FUNCTION_BLOCK FB_HMI_BUTTON
VAR_INPUT
    stColor : T_HMI_COLORS;
END_VAR
VAR_IN_OUT
    nActiveTab : INT;
    sActiveName : STRING;
END_VAR
VAR_OUTPUT
    sName : STRING;
    sIconName : STRING;
    nThisTab : INT;
    bActivated : BOOL;
    bNotActivated : BOOL;
    
    bIsNotGreen : BOOL;
    bIsNotRed : BOOL;
    bIsNotBlue : BOOL;
    bIsNotOrange : BOOL;
    bIsNotGray : BOOL;
END_VAR
VAR
    bDoActivate : BOOL;
    bPreviouslyActive : BOOL;
END_VAR

IF bDoActivate THEN
    nActiveTab := nThisTab;
    bDoActivate := FALSE;
END_IF

bActivated := nActiveTab = nThisTab;
bNotActivated := NOT bActivated;

IF bActivated AND NOT bPreviouslyActive THEN
    sActiveName := sName;
    bPreviouslyActive := TRUE;
END_IF

IF bNotActivated THEN
    bPreviouslyActive := FALSE;
END_IF

bIsNotRed    := stColor.bg <> E_HMI_Colors.RED;
bIsNotBlue   := stColor.bg <> E_HMI_Colors.BLUE;
bIsNotOrange := stColor.bg <> E_HMI_Colors.ORANGE;
bIsNotGray   := stColor.bg <> E_HMI_Colors.GRAY;
bIsNotGreen  := stColor.bg <> E_HMI_Colors.GREEN;

METHOD FB_init : BOOL
VAR_INPUT
	bInitRetains : BOOL; // if TRUE, the retain variables are initialized (warm start / cold start)
	bInCopyCode : BOOL;  // if TRUE, the instance afterwards gets moved into the copy code (online change)
    sName : STRING;
    sIconName : STRING;
    nThisTab : INT;
END_VAR
THIS^.sName := sName;
THIS^.sIconName := sIconName;
THIS^.nThisTab := nThisTab;
END_METHOD

METHOD M_SetIconName
VAR_INPUT
    sIconName : STRING;
END_VAR
THIS^.sIconName := sIconName;
END_METHOD

END_FUNCTION_BLOCK

(* stored: Version 1.1.0.1, ProductVersion 3.1.4024.14
   POU FB_HMI_BUTTON: Id {8312f969-1e2d-4234-8fb1-a5ec8ac8ee74}, SpecialFunc None
   Method FB_init: Id {09c2525c-94e5-4dbc-b816-3992467ecbb0}
   Method M_SetIconName: Id {045acce2-8b00-4ad1-a4e3-fbea920cbd17} *)
